{attribute 'linkalways'} 
{attribute 'no_explicit_call' := 'This FB is a CLASS and must be accessed using methods or properties'}
{attribute 'enable_dynamic_creation'}
FUNCTION_BLOCK Node_F_VN_AddToContainerElements_TcVnPoint2_LREAL EXTENDS VisionNode
VAR
    aValue : _TcVnPoint2_LREAL;
    ipContainer : _ITcVnContainer;
    hrPrev : _HRESULT(S_OK);
    hresult : _HRESULT(S_OK);
END_VAR

METHOD PUBLIC  Clone : I_Node
VAR
    pNode : POINTER TO Node_F_VN_AddToContainerElements_TcVnPoint2_LREAL;
END_VAR
pNode := __NEW(Node_F_VN_AddToContainerElements_TcVnPoint2_LREAL);
Clone := pNode^;
END_METHOD

METHOD FB_init : BOOL
VAR_INPUT
    bInitRetains : BOOL; // if TRUE, the retain variables are initialized (warm start / cold start)
    bInCopyCode : BOOL;  // if TRUE, the instance afterwards gets moved into the copy code (online change)
END_VAR
AddInput('aValue', aValue);
AddInput('ipContainer', ipContainer);
AddInput('hrPrev', hrPrev);
AddOutput('ipContainer', ipContainer);
AddOutput('hresult',hresult);
END_METHOD

METHOD PROTECTED OnExecute
hresult.Value := F_VN_AddToContainerElements_TcVnPoint2_LREAL(
    aValue := aValue.Value,
    ipContainer := ipContainer.Value,
    hrPrev:= hrPrev.Value);
END_METHOD

METHOD PUBLIC PreExecutionCheck
VAR_INPUT
    Check : I_PreExecutionChecks;
END_VAR
Check.IsTrue(ipContainer.IsValid, 'ipContainer must be a valid container');
Check.IsTrue(ipContainer.IsType(TC_GLOBAL_CONST_LIST.ContainerType_Vector_TcVnPoint2_LREAL), 'ipContainer contains incorrect type');
END_METHOD

END_FUNCTION_BLOCK

(* stored: Version 1.1.0.1, ProductVersion 3.1.4026.13
   POU Node_F_VN_AddToContainerElements_TcVnPoint2_LREAL: Id {e8cca6cd-0f84-4fa6-a0fd-823caae40b0d}, SpecialFunc None
   Folder Constructor: Id {c6492310-1f96-479b-a4c5-f0cc3d050386}
   Method Clone: Id {6d90025b-3319-4e50-a13c-2a0a40c652bc}
   Method FB_init: Id {de1d05a1-c8ff-4516-b35f-158523b03859}
   Method OnExecute: Id {3824c2c7-762b-4c5d-9f4b-adca084e4a9a}
   Method PreExecutionCheck: Id {7cdfffab-9729-492d-b81c-c4db8a3292d7} *)
